(* CoDeSys 2.3 export: FB_DECODE_FEDB.EXP *)

(* POU PGN FB/FB_DECODE_FEDB, ST *)
FUNCTION_BLOCK FB_DECODE_FEDB (*SPN 157 Engine Injector Metering Rail 1 Pressure*)
VAR_IN_OUT
	IN: ARRAY [0..7] OF USINT;
END_VAR
VAR_OUTPUT
	EngineInjectorMeteringRail1Pressure : REAL;

	Count : DWORD;
END_VAR
VAR
	Debug : BOOL;
	Buffer: ARRAY [0..7] OF USINT;
END_VAR
EngineInjectorMeteringRail1Pressure  := BUFFER_TO_REAL( pBuffer:= ADR(IN[2]), ByteSize := 2, Scale:= 0.00390625, Offset:= 0.0 );

Count := Count + 1;

IF Debug THEN MEMCPY(destAddr := ADR(Buffer), srcAddr := ADR(IN), n := 8); END_IF
END_FUNCTION_BLOCK
